// TIA Portal V16 export
// export: Created 2022-11-14T17:35:29.8929201Z, ExportSetting WithDefaults, DisplayName Totally Integrated Automation Portal, DisplayVersion V16, DisplayName TIA Portal Version Control Interface, DisplayVersion V16, DisplayName TIA Portal Openness, DisplayVersion V16, DisplayName STEP 7 Professional, DisplayVersion V16, DisplayName STEP 7 Safety, DisplayVersion V16, DisplayName WinCC Advanced, DisplayVersion V16
FUNCTION "FC43_PreCarriageTechnoplat" : Void   // FC43, LAD
TITLE = HS40 standard prestretch management
{ S7_Optimized_Access := 'FALSE' }
AUTHOR : Robopac
VERSION : 0.0
// stored: AutoNumber false, IsIECCheckEnabled false, SetENOAutomatically false, UDAEnableTagReadback false
BEGIN

REGION Network 1: Timer for prestretch restart
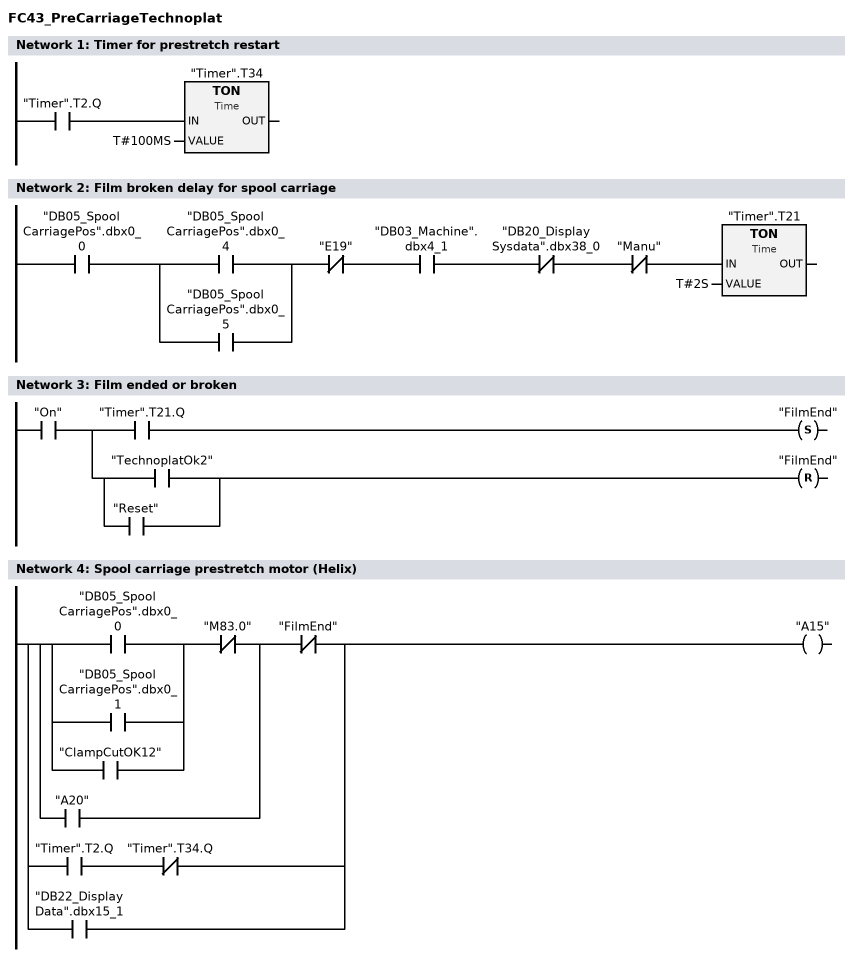
   "Timer".T34.TON(IN := "Timer".T2.Q, PT := T#100MS);   // TON coil
END_REGION

REGION Network 2: Film broken delay for spool carriage
   "Timer".T21.TON(IN := "DB05_SpoolCarriagePos".dbx0_0 AND ("DB05_SpoolCarriagePos".dbx0_4 OR "DB05_SpoolCarriagePos".dbx0_5) AND NOT "E19" AND "DB03_Machine".dbx4_1 AND NOT "DB20_DisplaySysdata".dbx38_0 AND NOT "Manu", PT := T#2S);   // TON coil
END_REGION

REGION Network 3: Film ended or broken
   RUNG wire#powerrail
      Contact( "On" )
      wire#w1
      Contact( "Timer".T21.Q )
      S_Coil( "FilmEnd" )
   END_RUNG
   RUNG wire#w1
      Contact( "TechnoplatOk2" )
      wire#w2
      R_Coil( "FilmEnd" )
   END_RUNG
   RUNG wire#w1
      Contact( "Reset" )
   END_RUNG wire#w2
   // the same network as SCL:
   IF "On" AND "Timer".T21.Q THEN "FilmEnd" := TRUE; END_IF;
   IF "On" AND ("TechnoplatOk2" OR "Reset") THEN "FilmEnd" := FALSE; END_IF;
END_REGION

REGION Network 4: Spool carriage prestretch motor (Helix)
   RUNG wire#powerrail
      Contact( "DB05_SpoolCarriagePos".dbx0_0 )
      wire#w1
      I_Contact( "M83.0" )
      wire#w2
      I_Contact( "FilmEnd" )
      wire#w3
      Coil( "A15" )
   END_RUNG
   RUNG wire#powerrail
      Contact( "DB05_SpoolCarriagePos".dbx0_1 )
   END_RUNG wire#w1
   RUNG wire#powerrail
      Contact( "ClampCutOK12" )
   END_RUNG wire#w1
   RUNG wire#powerrail
      Contact( "A20" )
   END_RUNG wire#w2
   RUNG wire#powerrail
      Contact( "Timer".T2.Q )
      I_Contact( "Timer".T34.Q )
   END_RUNG wire#w3
   RUNG wire#powerrail
      Contact( "DB22_DisplayData".dbx15_1 )
   END_RUNG wire#w3
   // the same network as SCL:
   "A15" := (((("DB05_SpoolCarriagePos".dbx0_0 OR "DB05_SpoolCarriagePos".dbx0_1 OR "ClampCutOK12") AND NOT "M83.0") OR "A20") AND NOT "FilmEnd") OR ("Timer".T2.Q AND NOT "Timer".T34.Q) OR "DB22_DisplayData".dbx15_1;
END_REGION
END_FUNCTION
